FUNCTION invMat2_1 : bool
VAR_IN_OUT CONSTANT
	mat :Mat2d;
END_VAR
VAR_IN_OUT
	invMat : Mat2d;
END_VAR
VAR
	matDet:LREAL;
END_VAR

matDet := mat[1,1]*mat[2,2]-mat[1,2]*mat[2,1];

IF ABS(matDet)<g_smallNum THEN
	invMat2 := FALSE;
	RETURN;
END_IF

invMat[1,1]:= mat[2,2]/matDet;
invMat[1,2]:= -mat[1,2]/matDet;
invMat[2,1]:= -mat[2,1]/matDet;
invMat[2,2]:= mat[1,1]/matDet;
 
invMat2:=TRUE;

END_FUNCTION

(* stored: Version 1.1.0.1, ProductVersion 3.1.4024.12
   POU invMat2_1: Id {06345110-d3ea-46ce-9bb6-f420ee50eb73}, SpecialFunc None *)
